TYPE (* A Template for a Data Type *)
  (* Version 0.0, 2020-04-28, 4DIAC-IDE, 4DIAC-Consortium *)
  (* ASN.1 tag APPLICATION 1 *)
  TemplateStruct : STRUCT
    MemberName : ANY_ELEMENTARY; (* Description *)
  END_STRUCT;
END_TYPE
